SUBAPPLICATION Uebung_028c3_AR (* Analog-Eingang Kalibrierung mit Adaptern INI und Hysterese-Regler am Ausgang und Display Anzeige *)
  (* Standard: 61499-2; Description: Copyright (c) 2026 Meisterschulen am Ostbahnhof This program and the accompanying materials are made available under the terms of the Eclipse Public License 2.0 which is available at https://www.eclipse.org/legal/epl-2.0/ SPDX-License-Identifier: EPL-2.0 *)
  (* Version 1.0, 2026-05-07, Franz Höpfinger, Meisterschulen am Ostbahnhof, initial API and implementation and/or initial documentation *)
  PACKAGE Uebungen;
  IMPORT Uebungen::const::UT::PWM::DefaultPool_PWM_Numeric::InputNumber_PWM_DUTY_OUT_N;
  IMPORT logiBUS::io::AI::logiBUS_AI::AnalogInput_I7;
  IMPORT logiBUS::io::DI::logiBUS_DI::Input_I1;
  IMPORT logiBUS::io::DI::logiBUS_DI::Input_I2;
  IMPORT logiBUS::io::DI::logiBUS_DI::Input_I3;
  IMPORT logiBUS::io::DI::logiBUS_DI_Events::BUTTON_SINGLE_CLICK;
  IMPORT logiBUS::io::DQ::logiBUS_DO::Output_Q1;
  IMPORT logiBUS::io::DQ::logiBUS_DO::Output_Q2;
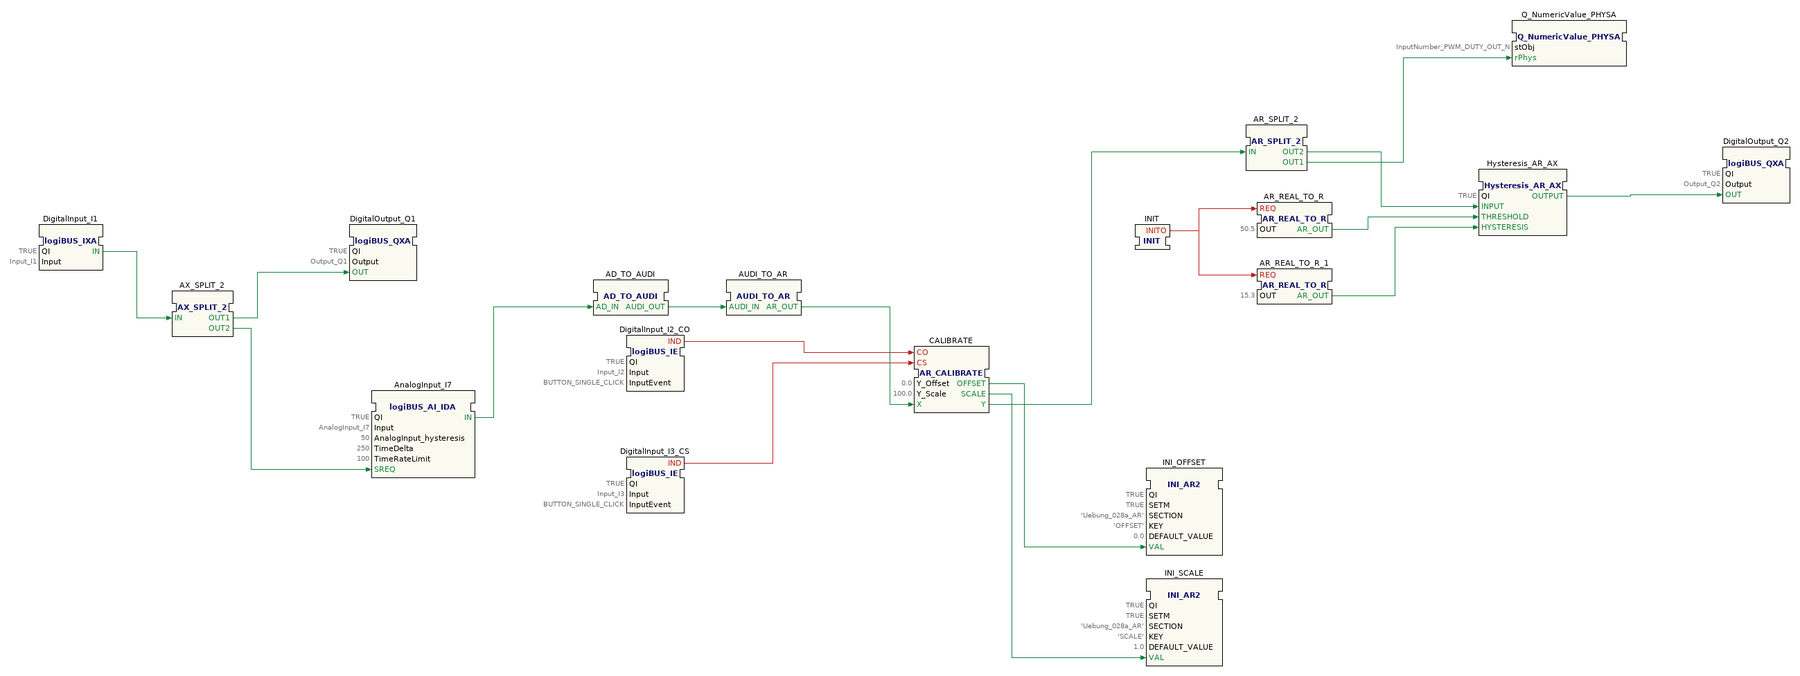
  (* WICHTIG ! Doppelte Konvertierung. ein AD_TO_AR wäre wie ein "reinterpret_cast" *)
  (* Beispiel: 0.0 => 0,5V 100.0 => 4,5V (Typ. Sensor Automotive) *)
  FBS
    DigitalInput_I1 : logiBUS::io::DI::logiBUS_IXA(QI := TRUE, Input := Input_I1);
    DigitalOutput_Q1 : logiBUS::io::DQ::logiBUS_QXA(QI := TRUE, Output := Output_Q1);
    AnalogInput_I7 : logiBUS::io::AI::logiBUS_AI_IDA(QI := TRUE, Input := AnalogInput_I7, AnalogInput_hysteresis := 50, TimeDelta := 250, TimeRateLimit := 100);
    CALIBRATE : adapter::Engineering::measurements::AR_CALIBRATE(Y_Offset := 0.0, Y_Scale := 100.0);
    INI_OFFSET : eclipse4diac::storage::INI_AR2(QI := TRUE, SETM := TRUE, SECTION := 'Uebung_028a_AR', KEY := 'OFFSET', DEFAULT_VALUE := 0.0);
    INI_SCALE : eclipse4diac::storage::INI_AR2(QI := TRUE, SETM := TRUE, SECTION := 'Uebung_028a_AR', KEY := 'SCALE', DEFAULT_VALUE := 1.0);
    DigitalInput_I2_CO : logiBUS::io::DI::logiBUS_IE(QI := TRUE, Input := Input_I2, InputEvent := BUTTON_SINGLE_CLICK);
    DigitalInput_I3_CS : logiBUS::io::DI::logiBUS_IE(QI := TRUE, Input := Input_I3, InputEvent := BUTTON_SINGLE_CLICK);
    AX_SPLIT_2 : adapter::events::unidirectional::AX_SPLIT_2;
    Hysteresis_AR_AX : logiBUS::signalprocessing::hysteresis::Hysteresis_AR_AX(QI := TRUE);
    AR_SPLIT_2 : adapter::events::unidirectional::AR_SPLIT_2;
    Q_NumericValue_PHYSA : isobus::UT::Q::Q_NumericValue_PHYSA(stObj := InputNumber_PWM_DUTY_OUT_N);
    AD_TO_AUDI : adapter::conversion::unidirectional::AD_TO_AUDI;
    AUDI_TO_AR : adapter::conversion::unidirectional::AUDI_TO_AR;
    DigitalOutput_Q2 : logiBUS::io::DQ::logiBUS_QXA(QI := TRUE, Output := Output_Q2);
    AR_REAL_TO_R : adapter::conversion::unidirectional::AR_REAL_TO_R(OUT := 50.5);
    AR_REAL_TO_R_1 : adapter::conversion::unidirectional::AR_REAL_TO_R(OUT := 15.3);
    INIT : iec61131::booleanOperators::INIT;
  END_FBS
  EVENT_CONNECTIONS
    INIT.INITO TO AR_REAL_TO_R.REQ;
    INIT.INITO TO AR_REAL_TO_R_1.REQ;
    DigitalInput_I2_CO.IND TO CALIBRATE.CO;
    DigitalInput_I3_CS.IND TO CALIBRATE.CS;
  END_CONNECTIONS
  ADAPTER_CONNECTIONS
    DigitalInput_I1.IN TO AX_SPLIT_2.IN;
    AnalogInput_I7.IN TO AD_TO_AUDI.AD_IN;
    AUDI_TO_AR.AR_OUT TO CALIBRATE.X;
    AX_SPLIT_2.OUT1 TO DigitalOutput_Q1.OUT;
    CALIBRATE.OFFSET TO INI_OFFSET.VAL;
    CALIBRATE.SCALE TO INI_SCALE.VAL;
    CALIBRATE.Y TO AR_SPLIT_2.IN;
    AR_SPLIT_2.OUT2 TO Hysteresis_AR_AX.INPUT;
    AR_SPLIT_2.OUT1 TO Q_NumericValue_PHYSA.rPhys;
    AD_TO_AUDI.AUDI_OUT TO AUDI_TO_AR.AUDI_IN;
    AX_SPLIT_2.OUT2 TO AnalogInput_I7.SREQ;
    Hysteresis_AR_AX.OUTPUT TO DigitalOutput_Q2.OUT;
    AR_REAL_TO_R.AR_OUT TO Hysteresis_AR_AX.THRESHOLD;
    AR_REAL_TO_R_1.AR_OUT TO Hysteresis_AR_AX.HYSTERESIS;
  END_CONNECTIONS
END_SUBAPPLICATION
